FUNCTION_BLOCK FB_Application
VAR_INPUT
END_VAR
VAR_OUTPUT
END_VAR
VAR
	safety : FB_Safety_module;
	tote_subsystem	: FB_Tote_Subsystem;
	light_tower	: FB_Light_tower_module;
END_VAR

safety();
light_tower();
tote_subsystem();

GVL.fb_mcp.lightTower := light_tower._lightTower;
GVL.fb_loading.lightTower	:= light_tower._lightTower;

END_FUNCTION_BLOCK

(* stored: Version 1.1.0.1, ProductVersion 3.1.4024.12
   POU FB_Application: Id {07911908-a847-4939-9523-bbe51254dbe7}, SpecialFunc None *)
